{attribute 'qualified_only'}
{attribute 'strict'}
TYPE E_JXCE1_GenericErrors :
(
	SPEED_SET_TOO_LOW := 1000,
	NEGATIVE_SPEED_USED := 1010,
	SET_POSITION_OUT_OF_STROKE_RANGE := 1100
);
END_TYPE

(* stored: Version 1.1.0.1, ProductVersion 3.1.4024.15
   DUT E_JXCE1_GenericErrors: Id {a03135b5-fb1b-052a-2ced-ba7c55cf4e4f} *)
